Staubli VAL3: extractCol.pgx

public program extractCol(num& x_nInput[] (dimensions=2), num x_nCol, num& x_nResult[])
  local num l_nCol
  local num l_nCounter
  local num l_nRow
begin

  resize(x_nResult,1,1)
  x_nResult = 0
  resize(x_nResult,1, size(x_nInput,1))

  l_nCounter = 0
  for l_nRow = 0 to size(x_nInput,1)-1
    x_nResult[l_nCounter] = x_nInput[l_nRow,x_nCol]
    l_nCounter = l_nCounter +1
  endFor

end
